INTERFACE IAssembly EXTENDS ZApplication.IUnit

END_INTERFACE

(* stored: Version 1.1.0.1
   Itf IAssembly: Id {dbe0929f-decf-46b0-916d-b95a28c0666d} *)
